// TwinCAT 3 PLC project PLC
// ProgramVersion: 3.1.4026.20
// CompilerDefines: VISU_USEPROPERTYINFO
// libraries:
//   SPT Base Types, * (Beckhoff Automation LLC)
//   SPT Components, * (Beckhoff Automation LLC)
//   SPT Diagnostic, * (Beckhoff Automation LLC)
//   SPT EtherCat, * (Beckhoff Automation LLC)
//   SPT Event Logger, * (Beckhoff Automation LLC)
//   SPT Motion Control, * (Beckhoff Automation LLC)
//   SPT Utilities, * (Beckhoff Automation LLC)
//   Tc2_MC2, * (Beckhoff Automation GmbH)
//   Tc2_MC2_Camming, * (Beckhoff Automation GmbH)
//   Tc2_Standard, * (Beckhoff Automation GmbH)
//   Tc2_System, * (Beckhoff Automation GmbH)
//   Tc2_Utilities, * (Beckhoff Automation GmbH)
//   Tc3_EventLogger, * (Beckhoff Automation GmbH)
//   Tc3_MC2_AdvancedHoming, * (Beckhoff Automation GmbH)
//   Tc3_McCollisionAvoidance, * (Beckhoff Automation GmbH)
//   Tc3_McCoordinatedMotion, * (Beckhoff Automation GmbH)
//   Tc3_PackML_V3, * (Beckhoff Automation GmbH)
// project tree:
//   / GlobalTextList.TcGTLO (not stored), PlcTask.TcTTO (not stored), VisualizationManager.TcVMO (not stored)
//   GVLs/ GVL.TcGVL (not stored)
//   POUs/EquipmentModules/CoupledMotion/ FB_CoupledMotion.TcPOU
//   POUs/ Machine.TcPOU, MAIN.TcPOU (not stored)
//   VISUs/ Visualization.TcVIS (not stored)
// real-time tasks:
//   TASK PlcTask: cycle T#1ms, priority 20, ADS port 350
//   TASK Job Task: cycle default, priority 32
// motion (NC):
//   TASK NC-Task 1 SAF: cycle T#2ms, priority 4, ADS port 501
//   TASK NC-Task 1 SVB: cycle T#10ms, priority 8, ADS port 511
//   AXIS PositionAxis (id 6)
//     General: UnitName=°
//     Dynamic: Acceleration=15000, Deceleration=15000, Jerk=131331.402
//     Velo: RefSearch=291.84756, RefSync=291.84756, SlowManual=1459.2378, FastManual=8755.4268, Fast=29184.756, Maximum=29184.756
//     OtherSettings: AllowMotionCmdToSlave=true
//     encoder EncType=8
//       EncPara: ScaleFactorNumerator=360, ScaleFactorDenominator=1048576, MaxCount=#xffffffff
//     drive DrvType=9
//       DrvPara: MaxCount=#xffffffff, DriveControlDWord=#x00030000
//         Analog: VeloReferenz=32103.2316, VeloScale=1.02400649589962, TorqueSetpointScale=10, ScaleFactorActTorque=0.1
//         TimeComp: TaskDelayCycles=1
//     controller CtrType=1
//       CtrPara: PriorControlFactor=1
//         PosDiffControl: Range=36
//         Observer: BandWidth=20
//   AXIS TorqueAxis (id 7)
//     General: UnitName=°
//     Dynamic: Acceleration=15000, Deceleration=15000, Jerk=131331.402
//     Velo: RefSearch=291.84756, RefSync=291.84756, SlowManual=1459.2378, FastManual=8755.4268, Fast=29184.756, Maximum=29184.756
//     OtherSettings: AllowMotionCmdToSlave=true
//     encoder EncType=8
//       EncPara: ScaleFactorNumerator=360, ScaleFactorDenominator=1048576, MaxCount=#xffffffff
//     drive DrvType=9
//       DrvPara: MaxCount=#xffffffff, DriveControlDWord=#x00030000
//         Analog: VeloReferenz=32103.2316, VeloScale=1.02400649589962, TorqueSetpointScale=10, ScaleFactorActTorque=0.1
//         TimeComp: TimeCompMode=1, TaskDelayCycles=1
//     controller CtrType=1
//       CtrPara: PriorControlFactor=1
//         Observer: BandWidth=20
// I/O:
//   DEVICE Device 3 (EtherCAT), AmsNetId 192.168.1.213.4.1
//     Drive 5 (AX5206-0000-0214) [AX5206-0000-0214 EtherCAT Drive (SoE, 2 Ch.)]
// variable links:
//   NC-Task 1 SAF/Axes/PositionAxis <-> Device 3 (EtherCAT)/Drive 5 (AX5206-0000-0214)
//     Drive/Inputs/In/nDataIn1 <-> AT 1/Following distance
//     Drive/Inputs/In/nDataIn3[0] <-> AT 1/Torque/force feedback value
//     Drive/Inputs/In/nDcOutputTime <-> InfoData/DcOutputShift
//     Drive/Inputs/In/nState1 <-> AT 1/Drive status word @bit 8
//     Drive/Inputs/In/nState2 <-> AT 1/Drive status word
//     Drive/Inputs/In/nState4 @bit 1 <-> WcState/InputToggle
//     Drive/Inputs/In/nState4 <-> WcState/WcState
//     Drive/Outputs/Out/nCtrl1 <-> MDT 1/Master control word @bit 8
//     Drive/Outputs/Out/nDataOut1 <-> MDT 1/Position command value
//     Drive/Outputs/Out/nDataOut4[0] <-> MDT 1/Torque/force command value
//     Drive/Outputs/Out/nDataOut5 <-> MDT 1/High velocity limit value
//     Drive/Outputs/Out/nDataOut6 <-> MDT 1/Low velocity limit value
//     Enc/Inputs/In/nDataIn1 <-> AT 1/Position feedback 1 value
//     Enc/Inputs/In/nDcInputTime <-> InfoData/DcInputShift
//     Enc/Inputs/In/nState4 @bit 1 <-> WcState/InputToggle
//     Enc/Inputs/In/nState4 <-> WcState/WcState
//   NC-Task 1 SAF/Axes/TorqueAxis <-> Device 3 (EtherCAT)/Drive 5 (AX5206-0000-0214)
//     Drive/Inputs/In/nDataIn1 <-> AT 2/Following distance
//     Drive/Inputs/In/nDataIn3[0] <-> AT 2/Torque/force feedback value
//     Drive/Inputs/In/nDcOutputTime <-> InfoData/DcOutputShift
//     Drive/Inputs/In/nState1 <-> AT 2/Drive status word @bit 8
//     Drive/Inputs/In/nState2 <-> AT 2/Drive status word
//     Drive/Inputs/In/nState4 @bit 1 <-> WcState/InputToggle
//     Drive/Inputs/In/nState4 <-> WcState/WcState
//     Drive/Outputs/Out/nCtrl1 <-> MDT 2/Master control word @bit 8
//     Drive/Outputs/Out/nDataOut1 <-> MDT 2/Position command value
//     Drive/Outputs/Out/nDataOut4[0] <-> MDT 2/Torque/force command value
//     Drive/Outputs/Out/nDataOut5 <-> MDT 2/High velocity limit value
//     Drive/Outputs/Out/nDataOut6 <-> MDT 2/Low velocity limit value
//     Enc/Inputs/In/nDataIn1 <-> AT 2/Position feedback 1 value
//     Enc/Inputs/In/nDcInputTime <-> InfoData/DcInputShift
//     Enc/Inputs/In/nState4 @bit 1 <-> WcState/InputToggle
//     Enc/Inputs/In/nState4 <-> WcState/WcState
//   PLC/PLC Instance <-> NC-Task 1 SAF/Axes/PositionAxis
//     PlcTask Inputs/MAIN.Machine.CoupledMotion.PositionAxis.BasicAxis._Axis.NcToPlc <-> Outputs/ToPlc
//     PlcTask Outputs/MAIN.Machine.CoupledMotion.PositionAxis.BasicAxis._Axis.PlcToNc <-> Inputs/FromPlc
//   PLC/PLC Instance <-> NC-Task 1 SAF/Axes/TorqueAxis
//     PlcTask Inputs/MAIN.Machine.CoupledMotion.TorqueAxis.BasicAxis._Axis.NcToPlc <-> Outputs/ToPlc
//     PlcTask Outputs/MAIN.Machine.CoupledMotion.TorqueAxis.BasicAxis._Axis.PlcToNc <-> Inputs/FromPlc

// ---- POUs/EquipmentModules/CoupledMotion/FB_CoupledMotion.TcPOU
FUNCTION_BLOCK FB_CoupledMotion EXTENDS FB_PackML_BaseModule
VAR
	PositionAxis	: FB_Component_BasicAxis;
	TorqueAxis		: FB_Component_BasicAxis;
	SetTorque		: REAL	:= 25;
	TorqueControl	: MC_TorqueControl;
	TON_Dwell		: TON;
END_VAR

//! @summary This method contains code which will execute when this PackML module is in the <b>Aborting</b> state
METHOD PROTECTED Aborting
VAR
	SubModulesReady : BOOL := TRUE;
END_VAR
CASE DescendantSequenceState OF
	0:
		NoStateTasksToComplete := FALSE;
		DescendantSequenceState := DescendantSequenceState + 10;

	10:
		IF PositionAxis.Disable() AND TorqueAxis.Disable() THEN
			StateTasksComplete 		:= TRUE;
			DescendantSequenceState := DescendantSequenceState + 10;
		END_IF

	//20:	

	20:
		StateTasksComplete := TRUE;
END_CASE

SUPER^.Aborting();
END_METHOD

//! @summary This method contains code which will execute when this PackML module is in the <b>Clearing</b> state
METHOD PROTECTED Clearing

(*! <description> <b>Note:</b> The <i>Clear</i> command can also be thought of as a <i>fault reset</i> depite the ambiguity in the naming of the <i>Reset</i> state. 
<table> 
	<tr>
		<th> Previous State </th>
		<th> Transition In </th>
		<th> Transition Out </th>
		<th> Next State  </th> 
	</tr>
	<tr>
		<td> Aborted </td>
		<td> Clear Command </td> 
		<td> State Complete </td>
		<td> Stopped </td> 
	</tr>
</table>
This method is called as required by <c>StateControl()</c>
</description> 

*)
// CASE _CurrentMode OF
// 	E_PMLUnitMode.ePMLUnitMode_Production:
		CASE DescendantSequenceState OF
			0: //Init
				NoStateTasksToComplete := FALSE;

				//Reset Axes and  CA Group
				PositionAxis.Reset();
				TorqueAxis.Reset();
				DescendantSequenceState := DescendantSequenceState + 10;

			10: // Done	
				StateTasksComplete := TRUE;
		END_CASE

// END_CASE

SUPER^.Clearing();
END_METHOD

METHOD CyclicLogic
VAR_INPUT
END_VAR
SUPER^.CyclicLogic();

TorqueControl(Axis := TorqueAxis.Axis);
TON_Dwell();
END_METHOD

//! @summary This method contains code which will execute when this PackML module is in the <b>Execute</b> state
METHOD PROTECTED Execute
VAR
	i : UDINT;
END_VAR
CASE _CurrentMode OF
	E_PMLUnitMode.Production:
		0:	PositionAxis.MoveAbsolute(360, TRUE);
			DescendantSequenceState	:= DescendantSequenceState + 10;
	
		10:	IF PositionAxis.InPosition AND PositionAxis.SetPosition > 350 THEN
				TON_Dwell.IN			:= TRUE;
				DescendantSequenceState	:= DescendantSequenceState + 10;
			END_IF
	
		20: IF TON_Dwell.Q THEN
				TON_Dwell.IN	:= FALSE;
				PositionAxis.MoveAbsolute(0, TRUE);
				DescendantSequenceState	:= DescendantSequenceState + 10;
			END_IF
	
		30:	IF PositionAxis.InPosition AND PositionAxis.SetPosition < 10 THEN
				TON_Dwell.IN			:= TRUE;
				DescendantSequenceState	:= DescendantSequenceState + 10;
			END_IF
	
		40: IF TON_Dwell.Q THEN
				TON_Dwell.IN	:= FALSE;
				PositionAxis.MoveAbsolute(360, TRUE);
				DescendantSequenceState	:= 10;
			END_IF

	E_PMLUnitMode.Manual:
		PositionAxis.Disable();

END_CASE
END_METHOD

(* Basic module initialization logic*)
METHOD PROTECTED Initialize : BOOL
Initialize := FALSE;
CASE DescendantSequenceState OF
	0:
		RegisterComponent(Component := PositionAxis);
		RegisterComponent(Component := TorqueAxis);
		DescendantSequenceState := DescendantSequenceState + 10;

	10:
		IF SUPER^.Initialize() THEN
			DescendantSequenceState := DescendantSequenceState + 10;
		END_IF

	20:
		Initialize := TRUE;
END_CASE
END_METHOD

METHOD PROTECTED Resetting
VAR_INST
END_VAR
// CASE _CurrentMode OF
// 	E_PMLUnitMode.ePMLUnitMode_Production:
		CASE DescendantSequenceState OF
			0: //Init
				NoStateTasksToComplete := FALSE;
				DescendantSequenceState := DescendantSequenceState + 10;

			10: //Enable Axes
				IF PositionAxis.Enable() AND TorqueAxis.Enable() THEN
					DescendantSequenceState := DescendantSequenceState + 10;
				END_IF

			// Home Axes (set current position to 0)
			20: // Home Right Axis
				IF PositionAxis.Home() and torqueAxis.Home() THEN
					DescendantSequenceState := DescendantSequenceState + 10;
				END_IF

			30: //Clearing complete
				StateTasksComplete := TRUE;

		END_CASE
// END_CASE

SUPER^.Resetting();
END_METHOD

METHOD PROTECTED Starting
//CASE _CurrentMode OF
//	E_PMLUnitMode.ePMLUnitMode_Production:
		CASE DescendantSequenceState OF
			0:
				NoStateTasksToComplete	:= FALSE;
				DescendantSequenceState := 10;

			10: //Set Axis Parameters
				PositionAxis.Velocity		:= 360;		TorqueAxis.Velocity			:= 360;
				PositionAxis.Acceleration	:= 720;		TorqueAxis.Acceleration		:= 720;
				PositionAxis.Deceleration	:= 720;		TorqueAxis.Deceleration		:= 720;
				PositionAxis.Jerk			:= 10000;	TorqueAxis.Jerk				:= 10000;

				TorqueControl.Execute			:= TRUE;
				TorqueControl.ContinuousUpdate	:= TRUE;
				TorqueControl.Relative			:= FALSE;
				TorqueControl.Torque			:= SetTorque;
				TorqueControl.TorqueRamp		:= 1;
				TorqueControl.VelocityLimitHigh	:= 360;
				TorqueControl.VelocityLimitLow	:= 360;	

				TON_Dwell.PT				:= t#250ms;
				DescendantSequenceState 	:= DescendantSequenceState + 10;
				StateTasksComplete 			:= TRUE;

			20: // Done
				NoStateTasksToComplete		:= TRUE;

		END_CASE

	//E_PMLUnitMode.ePMLUnitMode_Manual:
//END_CASE

SUPER^.Starting();
END_METHOD

METHOD PROTECTED Stopping
//CASE _CurrentMode OF
//	E_PMLUnitMode.ePMLUnitMode_Production:
		CASE DescendantSequenceState OF
			0:
				NoStateTasksToComplete	:= FALSE;
				DescendantSequenceState := 10;

			10: TorqueControl.Execute		:= FALSE;
				DescendantSequenceState 	:= DescendantSequenceState + 10;

			20: // Done
				NoStateTasksToComplete		:= TRUE;

		END_CASE

	//E_PMLUnitMode.ePMLUnitMode_Manual:
//END_CASE

SUPER^.Starting();
END_METHOD

END_FUNCTION_BLOCK

// ---- POUs/Machine.TcPOU
FUNCTION_BLOCK Machine EXTENDS FB_PackML_BaseModule
VAR
	CoupledMotion	: FB_CoupledMotion;
END_VAR

METHOD PROTECTED HMIPermissions
AllowHMIControl(TRUE);
END_METHOD

(* Basic module initialization logic*)
METHOD PROTECTED Initialize : BOOL
Initialize := FALSE;
CASE DescendantSequenceState OF
	0:
		RegisterSubmodule(SubModule	:= CoupledMotion);
		DescendantSequenceState := DescendantSequenceState + 10;

	10:
		IF SUPER^.Initialize() THEN
			Initialize := TRUE;
		END_IF
END_CASE
END_METHOD

END_FUNCTION_BLOCK
